/// Event structure
TYPE ST_EventOutput :
STRUCT
	/// INDEX in global event-Array
	nIdx				: INT;		
	sPriority			: WSTRING;	
	nPriorityColor		: DWORD;
	sPosition			: T_MaxString;
	sDescription		: T_MaxString;
	sRaiseInfo			: STRING;

END_STRUCT
END_TYPE

(* stored: Version 1.1.0.1
   DUT ST_EventOutput: Id {1e6d29e2-4794-4cc6-acff-be121e24a707} *)
